{attribute 'qualified_only'}
{attribute 'strict'}
TYPE E_PumpControlMode :
(
	OFF := 0,					
	CONST_SPEED := 1,				
	CONST_DIFFPRESS := 6,		
	VAR_DIFFPRESS := 7,
	NONE := 99
);
END_TYPE

(* stored: Version 1.1.0.1, ProductVersion 3.1.4024.4
   DUT E_PumpControlMode: Id {d21ee8f4-c506-48d1-99c0-11394e7d62ad} *)
